{attribute 'pack_mode' := '1'} 
TYPE ST_Beckhoff_4DI_4DO :
STRUCT
	bIn1	AT %Q* : BIT;
	bIn2	AT %Q* : BIT;
	bIn3	AT %Q* : BIT;
	bIn4	AT %Q* : BIT;	
	bOut1	AT %I* : BIT;
	bOut2	AT %I* : BIT;
	bOut3	AT %I* : BIT;
	bOut4	AT %I* : BIT;	
END_STRUCT
END_TYPE

(* stored: Version 1.1.0.1, ProductVersion 3.1.4024.12
   DUT ST_Beckhoff_4DI_4DO: Id {79ddcdea-b6f3-0bab-17ea-9615e6b489ae} *)
